Universal Robots PolyScope program: po.urp

Program po (installation=po directory=/programs/usbdisk_1 createdIn=5.17.3 lastSavedIn=5.17.3 robotSerialNumber=20245300973)
Calibrated DH parameters: a=[-0.000142, -0.107677, -0.213255, 0.000064, -0.000146, 0]; d=[0.15177, 74.572137, -73.839329, -0.601665, 0.085103, 0.092049]; alpha=[1.569409, -0.002935, 0.006027, 1.569361, -1.572417, 0]; deltaTheta=[0, -1.113565, 7.41746, -0.020708, -0.000001, 0]
InitVariablesNode
Robot Program (runOnlyOnce=false)
  MoveJ speed 60 deg/s, acceleration 80 deg/s^2 (useActiveTCP=true) feature=Base
    Waypoint Waypoint_1: TCP in base x=-137.5 y=-363.487 z=-152.745 mm, rx=-2.6415 ry=0.0001 rz=0 rad; joints [-90.832, -177.762, -67.031, -53.763, 89.815, 179.26] deg
  Wait Sleep waitTime=1
  URCap Save Image (Robotiq_Wrist_Camera, Robotiq Inc.) dataModel(saveImageModel=[{"saveDirectory":"/programs/usbdisk_0"}]); state(isChildrenLocked=true)
    URCap On Save Image success (Robotiq_Wrist_Camera, Robotiq Inc.)
      'Optional'
    URCap On Save Image fail (Robotiq_Wrist_Camera, Robotiq Inc.)
      'Optional'
  Wait Sleep waitTime=0.5
  Popup Message (haltProgram=false message=run matlab script inputType=Text)
  MoveJ speed 60 deg/s, acceleration 80 deg/s^2 (useActiveTCP=true) feature=Base
    Waypoint Waypoint_2: TCP in base x=-1.118 y=-223.69 z=693.497 mm, rx=-0.0053 ry=-2.224 rz=2.2142 rad; joints [0, -90, 0, -90, 0, 0] deg
  URCap External Control (External Control, FZI Research Center for Information Technology)
